Fanuc KAREL source: IO0202.KL

-- PROVISIONAL review KL for V940-1; original PC SHA256 e42818faf3a4d60758b5d6ad25eeef900cec2a240984973afa1286df8f0815a8
-- Incomplete behavior may be omitted. Consult companion uncertainty JSON. Do not deploy.
PROGRAM IO0202
%NOLOCKGROUP
-- UNRESOLVED_LOCAL_POOL 5 cells at code offset 13; source declarations unknown
-- DIRECT_LOCAL_WORD_ACCESS alone does not prove INTEGER, REAL, or BOOLEAN
BEGIN
  -- V9_ZERO_TABLE_METADATA_HINT layout=0002_ascii; no indexed target words; source/name/runtime held
  -- UNRESOLVED_PC offsets 0-18; opcodes 2B,2C,7B
  -- UNRESOLVED_PC offsets 23-30; opcodes 9D,23
  -- UNRESOLVED_PC offsets 35-49; opcodes 2E,22,9D,33,35
  -- UNRESOLVED_PC offsets 54-61; opcodes 9D,23
  -- UNRESOLVED_PC offsets 66-77; opcodes 2E,23
  -- UNRESOLVED_PC offsets 82-111; opcodes 27,27,9D,27,49,7E,AD,22,27,9D,31
  -- UNRESOLVED_PC offsets 116-120; opcodes 7F
  -- UNRESOLVED_PC offsets 125-129; opcodes 27,AA
  -- UNRESOLVED_PC offsets 134-138; opcodes 7F
END IO0202
